PROGRAM PRG_TM1K2_ATM
VAR
    {attribute 'pytmc' := 'pv: TM1K2:ATM'}
    {attribute 'TcLinkTo' := '.fbThermoCouple1.bError := TIIB[TM1K2-EL3314-E5]^TC Inputs Channel 1^Status^Error;
                              .fbThermoCouple1.bUnderrange := TIIB[TM1K2-EL3314-E5]^TC Inputs Channel 1^Status^Underrange;
                              .fbThermoCouple1.bOverrange := TIIB[TM1K2-EL3314-E5]^TC Inputs Channel 1^Status^Overrange;
                              .fbThermoCouple1.iRaw := TIIB[TM1K2-EL3314-E5]^TC Inputs Channel 1^Value;
                              .fbFlowMeter.iRaw := TIIB[AT1K2-EL3052-E8]^AI Standard Channel 1^Value

'} // TM1K2 shares the same cooling meter as AT1K2
    fbTM1K2: FB_TM1K2;

    fbStateSetup: FB_StateSetupHelper;
    stDefault: ST_PositionState := (
        fVelocity := 1,
        bMoveOk := TRUE,
        bValid := TRUE
    );
END_VAR


fbStateSetup(stPositionState:=stDefault, bSetDefault:=TRUE);

fbStateSetup(stPositionState:=fbTM1K2.stOut, fPosition:=-16.00, fDelta:=7, sPmpsState:='TM1K2:ATM-OUT');
fbStateSetup(stPositionState:=fbTM1K2.stTarget1, fPosition:=-39.124, fDelta:=7, sPmpsState:='TM1K2:ATM-TARGET1');
fbStateSetup(stPositionState:=fbTM1K2.stTarget2, fPosition:=-53.5, fDelta:=7, sPmpsState:='TM1K2:ATM-TARGET2');
fbStateSetup(stPositionState:=fbTM1K2.stTarget3, fPosition:=-67.874, fDelta:=7, sPmpsState:='TM1K2:ATM-TARGET3');
fbStateSetup(stPositionState:=fbTM1K2.stTarget4, fPosition:=-82.25, fDelta:=7, sPmpsState:='TM1K2:ATM-TARGET4');
fbStateSetup(stPositionState:=fbTM1K2.stTarget5, fPosition:=-96.623, fDelta:=7, sPmpsState:='TM1K2:ATM-TARGET5');
fbStateSetup(stPositionState:=fbTM1K2.stTarget6, fPosition:=-114.5, fDelta:=7, sPmpsState:='TM2K2:ATM-DIODE');

fbTM1K2(
    fbFFHWO := GVL.fbFastFaultOutput2,
    fbArbiter := GVL.fbArbiter2,
    stYStage := Main.M9,
    stXStage := Main.M10,
    sDeviceName := 'TM1K2:ATM',
    sTransitionKey := 'TM1K2:ATM-TRANSITION',
    bEnableMotion := TRUE,
    bEnableBeamParams := TRUE,
    bEnablePositionLimits := TRUE,
);

END_PROGRAM

(* stored: Version 1.1.0.1, ProductVersion 3.1.4024.12
   POU PRG_TM1K2_ATM: Id {c02e8350-6bfd-4c3f-8509-cf01c04221fa}, SpecialFunc None *)
